Staubli VAL3: BytesToS16.pgx

program BytesToS16(num hByte, num lByte, num& result)
begin
//*******************************************************************************
//*   ______
//*  / _____) /|
//* | |      / /
//* | | /\  / /
//* | | \ \/ /  _      Copyright (c) KEOLABS, 2016
//* | |  \__/  | |        http://www.keolabs.com
//* | |________| |
//*  \__________/
//*
//********************************************************************************
//*@file          : BytesToS16
//*@author        : Yves Ragot
//*@version       : $Id: BytesToS16.pgx 1191 2016-10-05 15:10:08Z yves $
//*@brief         : convert 2 bytes into signed 16 bits word
//*
//*******************************************************************************/

  if (hByte < 128)
    result = (hByte * 256) + lByte
  else
    result = ((hByte * 256) + lByte) - 65536
  endIf

end
